// TIA Portal V17 export
// export: Created 2025-03-05T08:00:00.1041706Z, ExportSetting WithDefaults, DisplayName Totally Integrated Automation Portal, DisplayVersion V17 Update 8, DisplayName TIA Portal Openness, DisplayVersion V17 Update 8, DisplayName TIA Portal Version Control Interface, DisplayVersion V17, DisplayName SINAMICS Startdrive Advanced, DisplayVersion V17 SP2, DisplayName SINAMICS Startdrive G110M, G120, G120C, G120D, G120P, G115D, DisplayVersion V17 SP2, DisplayName SINAMICS Startdrive G130, G150, S120, S150, SINAMICS MV, S210, DisplayVersion V17 SP2, DisplayName STEP 7 Professional, DisplayVersion V17 Update 8, DisplayName SINUMERIK ONE STEP 7 Toolbox, DisplayVersion V17 Update 12, DisplayName SINUMERIK 840D sl STEP 7 Toolbox, DisplayVersion V17 Update 12, DisplayName STEP 7 Safety, DisplayVersion V17 Update 6, DisplayName WinCC Advanced, DisplayVersion V17 Update 8
FUNCTION "FC2000_MACHINE_MODES" : Void   // FC2000, LAD
{ S7_Optimized_Access := 'FALSE' }
AUTHOR : ETXETAR
VERSION : 1.0
// stored: AutoNumber false, IsIECCheckEnabled false, SetENOAutomatically false, UDAEnableTagReadback false
BEGIN

REGION Network 1: OPTIONS OFF
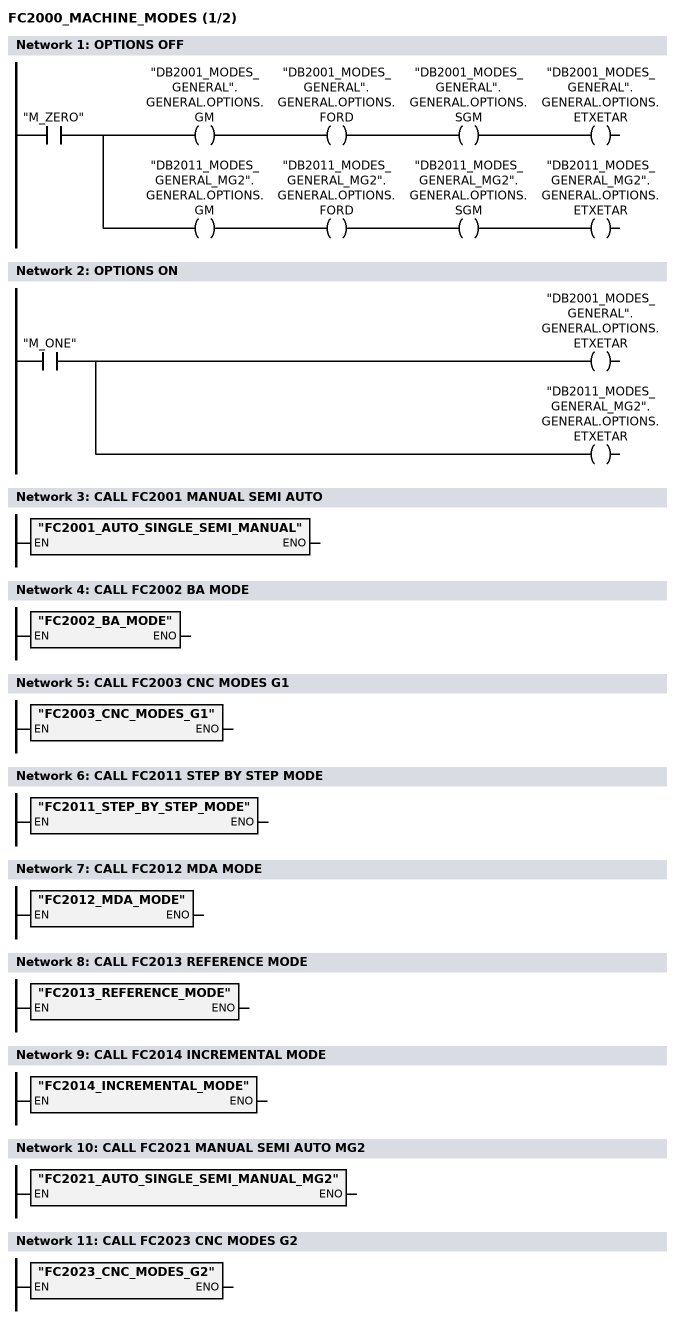
   RUNG wire#powerrail
      Contact( "M_ZERO" )
      wire#w1
      Coil( "DB2001_MODES_GENERAL".GENERAL.OPTIONS.GM )
      Coil( "DB2001_MODES_GENERAL".GENERAL.OPTIONS.FORD )
      Coil( "DB2001_MODES_GENERAL".GENERAL.OPTIONS.SGM )
      Coil( "DB2001_MODES_GENERAL".GENERAL.OPTIONS.ETXETAR )
   END_RUNG
   RUNG wire#w1
      Coil( "DB2011_MODES_GENERAL_MG2".GENERAL.OPTIONS.GM )
      Coil( "DB2011_MODES_GENERAL_MG2".GENERAL.OPTIONS.FORD )
      Coil( "DB2011_MODES_GENERAL_MG2".GENERAL.OPTIONS.SGM )
      Coil( "DB2011_MODES_GENERAL_MG2".GENERAL.OPTIONS.ETXETAR )
   END_RUNG
   // the same network as SCL:
   "DB2001_MODES_GENERAL".GENERAL.OPTIONS.GM := "M_ZERO";
   "DB2001_MODES_GENERAL".GENERAL.OPTIONS.FORD := "M_ZERO";
   "DB2001_MODES_GENERAL".GENERAL.OPTIONS.SGM := "M_ZERO";
   "DB2001_MODES_GENERAL".GENERAL.OPTIONS.ETXETAR := "M_ZERO";
   "DB2011_MODES_GENERAL_MG2".GENERAL.OPTIONS.GM := "M_ZERO";
   "DB2011_MODES_GENERAL_MG2".GENERAL.OPTIONS.FORD := "M_ZERO";
   "DB2011_MODES_GENERAL_MG2".GENERAL.OPTIONS.SGM := "M_ZERO";
   "DB2011_MODES_GENERAL_MG2".GENERAL.OPTIONS.ETXETAR := "M_ZERO";
END_REGION

REGION Network 2: OPTIONS ON
   RUNG wire#powerrail
      Contact( "M_ONE" )
      wire#w1
      Coil( "DB2001_MODES_GENERAL".GENERAL.OPTIONS.ETXETAR )
   END_RUNG
   RUNG wire#w1
      Coil( "DB2011_MODES_GENERAL_MG2".GENERAL.OPTIONS.ETXETAR )
   END_RUNG
   // the same network as SCL:
   "DB2001_MODES_GENERAL".GENERAL.OPTIONS.ETXETAR := "M_ONE";
   "DB2011_MODES_GENERAL_MG2".GENERAL.OPTIONS.ETXETAR := "M_ONE";
END_REGION

REGION Network 3: CALL FC2001 MANUAL SEMI AUTO
   RUNG wire#powerrail
      "FC2001_AUTO_SINGLE_SEMI_MANUAL"()
   END_RUNG
   // the same network as SCL:
   "FC2001_AUTO_SINGLE_SEMI_MANUAL"();
END_REGION

REGION Network 4: CALL FC2002 BA MODE
   RUNG wire#powerrail
      "FC2002_BA_MODE"()
   END_RUNG
   // the same network as SCL:
   "FC2002_BA_MODE"();
END_REGION

REGION Network 5: CALL FC2003 CNC MODES G1
   RUNG wire#powerrail
      "FC2003_CNC_MODES_G1"()
   END_RUNG
   // the same network as SCL:
   "FC2003_CNC_MODES_G1"();
END_REGION

REGION Network 6: CALL FC2011 STEP BY STEP MODE
   RUNG wire#powerrail
      "FC2011_STEP_BY_STEP_MODE"()
   END_RUNG
   // the same network as SCL:
   "FC2011_STEP_BY_STEP_MODE"();
END_REGION

REGION Network 7: CALL FC2012 MDA MODE
   RUNG wire#powerrail
      "FC2012_MDA_MODE"()
   END_RUNG
   // the same network as SCL:
   "FC2012_MDA_MODE"();
END_REGION

REGION Network 8: CALL FC2013 REFERENCE MODE
   RUNG wire#powerrail
      "FC2013_REFERENCE_MODE"()
   END_RUNG
   // the same network as SCL:
   "FC2013_REFERENCE_MODE"();
END_REGION

REGION Network 9: CALL FC2014 INCREMENTAL MODE
   RUNG wire#powerrail
      "FC2014_INCREMENTAL_MODE"()
   END_RUNG
   // the same network as SCL:
   "FC2014_INCREMENTAL_MODE"();
END_REGION

REGION Network 10: CALL FC2021 MANUAL SEMI AUTO MG2
   RUNG wire#powerrail
      "FC2021_AUTO_SINGLE_SEMI_MANUAL_MG2"()
   END_RUNG
   // the same network as SCL:
   "FC2021_AUTO_SINGLE_SEMI_MANUAL_MG2"();
END_REGION

REGION Network 11: CALL FC2023 CNC MODES G2
   RUNG wire#powerrail
      "FC2023_CNC_MODES_G2"()
   END_RUNG
   // the same network as SCL:
   "FC2023_CNC_MODES_G2"();
END_REGION

REGION Network 12: CALL FC2025 MDA MODE MG2
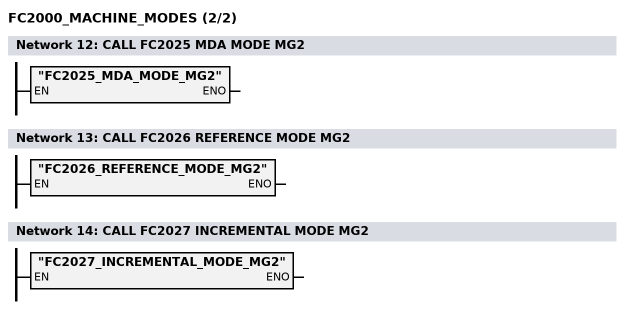
   RUNG wire#powerrail
      "FC2025_MDA_MODE_MG2"()
   END_RUNG
   // the same network as SCL:
   "FC2025_MDA_MODE_MG2"();
END_REGION

REGION Network 13: CALL FC2026 REFERENCE MODE MG2
   RUNG wire#powerrail
      "FC2026_REFERENCE_MODE_MG2"()
   END_RUNG
   // the same network as SCL:
   "FC2026_REFERENCE_MODE_MG2"();
END_REGION

REGION Network 14: CALL FC2027 INCREMENTAL MODE MG2
   RUNG wire#powerrail
      "FC2027_INCREMENTAL_MODE_MG2"()
   END_RUNG
   // the same network as SCL:
   "FC2027_INCREMENTAL_MODE_MG2"();
END_REGION
END_FUNCTION
